TYPE ST_StewartFeedback :
STRUCT
	eta: ARRAY[0..5] OF LREAL;
	eta_t: ARRAY[0..5] OF LREAL;
	eta_tt: ARRAY[0..5] OF LREAL;
END_STRUCT
END_TYPE

(* stored: Version 1.1.0.1, ProductVersion 3.1.4022.7
   DUT ST_StewartFeedback: Id {9b35b3d5-cd69-4c2c-bbf4-f9f9046d7699} *)
